FUNCTION_BLOCK FB_LimitLookup
VAR_INPUT
    fEnergy : LREAL;
END_VAR
VAR_OUTPUT
    bEnergyInTable : BOOL;
    fLow : LREAL;
    fHigh : LREAL;
END_VAR
VAR
    (* TC version doesn't appear to support dynamic arrays here *)
    (* falling back to pointer-handling; sorry! *)
    stRow : POINTER TO ST_TableRow;
    stNextRow : POINTER TO ST_TableRow;
    iRowCount : UINT;
    iRowIdx : UINT;
    fSlope : LREAL;
    fEnergyDelta : LREAL;
    iLensIdx: INT;
END_VAR

iLensIdx := F_GetXRTLensIndex();

IF iLensIdx = 1 THEN
    stRow := ADR(fbEnergyTables.stLENS1_750);
    iRowCount := SIZEOF(fbEnergyTables.stLENS1_750) / SIZEOF(ST_TableRow);
ELSIF iLensIdx = 2 THEN
    stRow := ADR(fbEnergyTables.stLENS2_428);
    iRowCount := SIZEOF(fbEnergyTables.stLENS2_428) / SIZEOF(ST_TableRow);
ELSIF iLensIdx = 3 THEN
    stRow := ADR(fbEnergyTables.stLENS3_333);
    iRowCount := SIZEOF(fbEnergyTables.stLENS3_333) / SIZEOF(ST_TableRow);
ELSE
    stRow := ADR(fbEnergyTables.stNO_LENS);
    iRowCount := SIZEOF(fbEnergyTables.stNO_LENS) / SIZEOF(ST_TableRow);
END_IF

fLow := 0.0;
fHigh := 0.0;
bEnergyInTable := FALSE;

IF fEnergy < stRow^.fEnergy THEN
    RETURN;
END_IF

FOR iRowIdx := 0 TO iRowCount - 2
DO
(*
 result->energy = find_energy;
 double slope = (rows[upper_idx].low - rows[lower_idx].low) / delta_energy;
 result->low = rows[lower_idx].low + slope * (find_energy - rows[lower_idx].energy);

 slope = (rows[upper_idx].high - rows[lower_idx].high) / delta_energy;
 result->high = rows[lower_idx].high + slope * (find_energy - rows[lower_idx].energy);
*)
    stNextRow := ADR(stRow[1]);
    IF fEnergy >= stRow^.fEnergy AND fEnergy <= stNextRow^.fEnergy THEN
        fEnergyDelta := stNextRow^.fEnergy - stRow^.fEnergy;
        IF fEnergyDelta > 0.0 THEN
            bEnergyInTable := TRUE;
            // Interpolate between the points
            fSlope := (stNextRow^.fLow - stRow^.fLow) / fEnergyDelta;
            fLow := stRow^.fLow + fSlope * (fEnergy - stRow^.fEnergy);

            fSlope := (stNextRow^.fHigh - stRow^.fHigh) / fEnergyDelta;
            fHigh := stRow^.fHigh + fSlope * (fEnergy - stRow^.fEnergy);
        END_IF
        RETURN;
    END_IF
    stRow := stNextRow;
END_FOR

END_FUNCTION_BLOCK

(* stored: Version 1.1.0.1, ProductVersion 3.1.4018.10
   POU FB_LimitLookup: Id {d2a23f8c-7f59-4e9d-888f-ed774cd15cbd}, SpecialFunc None *)
